(* CODESYS project untitled1.library
   Placeholder: TwinCAT_LIB
   Title: TwinCAT_LIB
   Version: 1.65
   Description: Baisc library's for s88 programming
   Company: Farnwood Engineering

Project tree, tasks and I/O mapping:
  libraries: Tc2_Standard, * (Beckhoff Automation GmbH); Tc2_System, * (Beckhoff Automation GmbH); Tc3_Module, * (Beckhoff Automation GmbH)
  DUTs/
  GVLs/
    POUs/
      LIB/
        1. Control Modules/
          1. DEV_Base/
            function block FB_DeviceBase [ST]
            data type stDevBase
          2. DEV_AnaIn/
            function block FB_DEV_AnaIn [ST]
            interface ITF_DEV_AnaIn
          3. DEV_DigIn/
            function block FB_DEV_DigIn [ST]: FB_init, Force, ResetForce, ActualValue, FallingEdge, RisingEdge
            interface ITF_DigIn: FB_init, Force, ResetForce, ActualValue, FallingEdge, RisingEdge
          4. DEV_Valve/
            ENUMs/
              data type E_ValveState
            STRUCTs/
              data type stDevValve
            function block DEV_Valve [ST]: _FExceptions, _StHmi, Close, Open, Reset, SetMode, ActualState, EmergencyStatus, OperatingMode
            interface ITF_Valve: Close, Open, Reset, SetMode, ActualState, EmergencyStatus, OperatingMode
          5. DEV_ControlValve/
            ENUMs/
              data type E_CtrlValveState
            STRUCTs/
            function block DEV_CtrlValve [ST]: EmergencyStatus, OperatingMode, OutputValue, Reset, SetMode, SetValue
            interface ITF_ControlValve: Reset, SetMode, SetValue, EmergencyStatus, OperatingMode, OutputValue
          6. DEV_Motor/
            ENUMs/
              data type E_MotorState
            STRUCTs/
            interface ITF_Motor: Auto, Manueel, Reset, Richting_L, Richting_R, Start, Stop, Toerental, ActualState, Error_State, State
          7. DEV_ControlMotor/
          ENUMs/
            data type E_OperationMode
          function block FB_Devices [ST]
        2. Equipment Modules/
          1. FB_Base/
            function block FB_EMbase [ST]
            data type stEMbase
          2. EM_Machine_PackML/
            data type E_State_PackML
            function block FB_Machine_PackML [ST]: Abort, Aborting_SC, Clear, Clearing_SC, Completing_SC, Execute_SC, Hold, Holding_SC, Reset, Resetting_SC, Start, Starting_SC, Stop, Stopping_SC, Suspend, Suspending_SC, Unhold, Unholding_SC, Unsuspend, Unsuspending_SC, State, FB_init, ZeroAllVar
            interface ITF_PackML: Abort, Aborting_SC, Clear, Clearing_SC, Completing_SC, Execute_SC, Hold, Holding_SC, Reset, Resetting_SC, Start, Starting_SC, Stop, Stopping_SC, Suspend, Suspending_SC, Unhold, Unholding_SC, Unsuspend, Unsuspending_SC, ZeroAllVar, State, FB_init
            data type STRUCT_Machine_PackML
          2. EM_Transport/
            Enums/
            Structs/
              1. CS/
                data type EM_Transport_CS
              2. HMI/
                data type EM_Transport_HMI
              3. STS/
                data type EM_Transport_STS
              4. ALM/
                data type EM_Transport_ALM
              5. WRN/
                data type EM_Transport_WRN
              6. PAR/
                data type EM_Transport_PAR
              7. SIM/
                data type EM_Transport_SIM
              data type STRUCT_EM_Transport
            function block EM_Transport [ST]: Abort, Clear, Reset, Start, Stop, Auto, Manueel, RPM, State, Tag, ZeroAllVar
            interface ITF_EM_Transport: Abort, Reset, Start, Stop, Auto, Manueel, RPM, State, Tag, ZeroAllVar
          3. EM_Transport_Mechanische_Stop/
            Enums/
              data type E_Mechanische_Stop
            Structs/
              1. CS/
                data type EM_Transport_Mechanische_Stop_CS
              2. HMI/
                data type EM_Transport_Mechanische_Stop_HMI
              3. STS/
                data type EM_Transport_Mechanische_Stop_STS
              4. ALM/
                data type EM_Transport_Mechanische_Stop_ALM
              5. WRN/
                data type EM_Transport_Mechanische_Stop_WRN
              6. PAR/
                data type EM_Transport_Mechanische_Stop_PAR
              7. SIM/
                data type EM_Transport_Mechanische_Stop_SIM
              data type STRUCT_EM_Mechanische_Stop
            function block EM_Transport_Mechanische_Stop [ST]: Close, Open, Stop_State, ZeroAllValues
            interface ITF_EM_Transport_Mechanische_Stop: Close, Open, Stop_State, ZeroAllValues
        3. Units/
          1. UN_Base/
            function block FB_UN_base [ST]
            data type stUNbase
        4. Management layer/
          FB_Alarmhandler/
        FUN/
          function PackML [ST]
          data type STRUCT_PackML
      program MAIN [ST]
  Version/
    global variables Global_Version
  VISUs/
*)

// GVLs/POUs/LIB/1. Control Modules/1. DEV_Base/stDevBase
TYPE stDevBase :
STRUCT
	sTagName : STRING;
	sDescription : STRING;
END_STRUCT
END_TYPE

// GVLs/POUs/LIB/1. Control Modules/4. DEV_Valve/ENUMs/E_ValveState
{attribute 'qualified_only'}
{attribute 'strict'}
TYPE E_ValveState :
(
	Unknown := 0,
	Open := 1,
	Closed := 2,
	Opening := 3,
	Closing := 4,
	Error := -1
);
END_TYPE

// GVLs/POUs/LIB/1. Control Modules/4. DEV_Valve/STRUCTs/stDevValve
TYPE stDevValve :
STRUCT
	//Input to HMI
	bGetHmiError : BOOL;  //True = error
	bGetHmiStatus : BOOL; //True = Open || False = Closed
	eGetState : E_ValveState;
	eGetMode : E_OperationMode;
	
	//Output from HMI
	eSetMode : E_OperationMode; 
END_STRUCT
END_TYPE

// GVLs/POUs/LIB/1. Control Modules/5. DEV_ControlValve/ENUMs/E_CtrlValveState
{attribute 'qualified_only'}
{attribute 'strict'}
TYPE E_CtrlValveState :
(
	Unknown := 0,
	InPosition := 1,
	Moving := 2,
	Error := -1
);
END_TYPE

// GVLs/POUs/LIB/1. Control Modules/6. DEV_Motor/ENUMs/E_MotorState
{attribute 'qualified_only'}
{attribute 'strict'}
TYPE E_MotorState :
(
	Unknown := 0,
	Running := 1,
	Stalled := 2,
	SpeedingUp := 3,
	SpeedingDown := 4,
	Error := -1
);
END_TYPE

// GVLs/POUs/LIB/1. Control Modules/ENUMs/E_OperationMode
{attribute 'qualified_only'}
{attribute 'strict'}
TYPE E_OperationMode :
(
	Off := 0,
	Manual := 1,
	Automatic := 2
);
END_TYPE

// GVLs/POUs/LIB/2. Equipment Modules/1. FB_Base/stEMbase
TYPE stEMbase :
STRUCT
	sTagName : STRING;
	sDescription : STRING;
END_STRUCT
END_TYPE

// GVLs/POUs/LIB/2. Equipment Modules/2. EM_Machine_PackML/E_State_PackML
{attribute 'qualified_only'}
{attribute 'strict'}
TYPE E_State_PackML :
(
	IDLE	:= 0,
	STARTING,
	EXECUTE,
	COMPLETING,
	COMPLETE,
	RESETTING,
	HOLDING,
	HELD,
	UNHOLDING,
	SUSPENDING,
	SUSPENDED,
	UNSUSPENDING,
	ABORTING,
	ABORTED,
	CLEARING,
	STOPPING,
	STOPPED
);
END_TYPE

// GVLs/POUs/LIB/2. Equipment Modules/2. EM_Machine_PackML/STRUCT_Machine_PackML
TYPE STRUCT_Machine_PackML :
STRUCT
	//Properties
	State 			: E_State_PackML;
	//Methods
   	Abort 			: BOOL;
	Aborting_SC 	: BOOL;
	Clear 			: BOOL;
	Clearing_SC 	: BOOL;
	Execute_SC 		: BOOL;
	Completing_SC	: BOOL;
	Hold 			: BOOL;
	Holding_SC 		: BOOL;
	Reset 			: BOOL;
	Resetting_SC 	: BOOL;
	Start 			: BOOL;
	Starting_SC 	: BOOL;
	Stop 			: BOOL;
	Stopping_SC 	: BOOL;
	Suspend 		: BOOL;
	Suspending_SC 	: BOOL;
	Unhold 			: BOOL;
	Unholding_SC 	: BOOL;
	Unsuspend 		: BOOL;
	Unsuspending_SC : BOOL;
END_STRUCT
END_TYPE

// GVLs/POUs/LIB/2. Equipment Modules/2. EM_Transport/Structs/1. CS/EM_Transport_CS
TYPE EM_Transport_CS :
STRUCT
	Start		: BOOL;
	Stop		: BOOL;
	Reset		: BOOL;
	Abort		: BOOL;
	Auto		: BOOL;
	Manueel		: BOOL;
END_STRUCT
END_TYPE

// GVLs/POUs/LIB/2. Equipment Modules/2. EM_Transport/Structs/2. HMI/EM_Transport_HMI
TYPE EM_Transport_HMI :
STRUCT
	Start		: BOOL;
	Stop		: BOOL;
	Reset		: BOOL;
	Abort		: BOOL;
	Auto		: BOOL;
	Manueel		: BOOL;
END_STRUCT
END_TYPE

// GVLs/POUs/LIB/2. Equipment Modules/2. EM_Transport/Structs/3. STS/EM_Transport_STS
TYPE EM_Transport_STS :
STRUCT
	Tag				: STRING;
	State 			: E_State_PackML;
	Manueel			: BOOL;
	Auto			: BOOL;
END_STRUCT
END_TYPE

// GVLs/POUs/LIB/2. Equipment Modules/2. EM_Transport/Structs/4. ALM/EM_Transport_ALM
TYPE EM_Transport_ALM :
STRUCT
END_STRUCT
END_TYPE

// GVLs/POUs/LIB/2. Equipment Modules/2. EM_Transport/Structs/5. WRN/EM_Transport_WRN
TYPE EM_Transport_WRN :
STRUCT
END_STRUCT
END_TYPE

// GVLs/POUs/LIB/2. Equipment Modules/2. EM_Transport/Structs/6. PAR/EM_Transport_PAR
TYPE EM_Transport_PAR :
STRUCT
END_STRUCT
END_TYPE

// GVLs/POUs/LIB/2. Equipment Modules/2. EM_Transport/Structs/7. SIM/EM_Transport_SIM
TYPE EM_Transport_SIM :
STRUCT
END_STRUCT
END_TYPE

// GVLs/POUs/LIB/2. Equipment Modules/2. EM_Transport/Structs/STRUCT_EM_Transport
TYPE STRUCT_EM_Transport :
STRUCT
	CS	: EM_Transport_CS;
	HMI	: EM_Transport_HMI;
	STS	: EM_Transport_STS;
	ALM	: EM_Transport_ALM;
	WRN	: EM_Transport_WRN;
	PAR	: EM_Transport_PAR;
	SIM	: EM_Transport_SIM;	
END_STRUCT
END_TYPE

// GVLs/POUs/LIB/2. Equipment Modules/3. EM_Transport_Mechanische_Stop/Enums/E_Mechanische_Stop
{attribute 'qualified_only'}
{attribute 'strict'}
TYPE E_Mechanische_Stop :
(
	enum_member := 0
);
END_TYPE

// GVLs/POUs/LIB/2. Equipment Modules/3. EM_Transport_Mechanische_Stop/Structs/1. CS/EM_Transport_Mechanische_Stop_CS
TYPE EM_Transport_Mechanische_Stop_CS :
STRUCT
	Start		: BOOL;
	Stop		: BOOL;
	Reset		: BOOL;
	Abort		: BOOL;
	Auto		: BOOL;
	Manueel		: BOOL;
END_STRUCT
END_TYPE

// GVLs/POUs/LIB/2. Equipment Modules/3. EM_Transport_Mechanische_Stop/Structs/2. HMI/EM_Transport_Mechanische_Stop_HMI
TYPE EM_Transport_Mechanische_Stop_HMI :
STRUCT
	Start		: BOOL;
	Stop		: BOOL;
	Reset		: BOOL;
	Abort		: BOOL;
	Auto		: BOOL;
	Manueel		: BOOL;
END_STRUCT
END_TYPE

// GVLs/POUs/LIB/2. Equipment Modules/3. EM_Transport_Mechanische_Stop/Structs/3. STS/EM_Transport_Mechanische_Stop_STS
TYPE EM_Transport_Mechanische_Stop_STS :
STRUCT
	Tag				: STRING;
	State 			: E_Mechanische_Stop;
	Manueel			: BOOL;
	Auto			: BOOL;
END_STRUCT
END_TYPE

// GVLs/POUs/LIB/2. Equipment Modules/3. EM_Transport_Mechanische_Stop/Structs/4. ALM/EM_Transport_Mechanische_Stop_ALM
TYPE EM_Transport_Mechanische_Stop_ALM :
STRUCT
END_STRUCT
END_TYPE

// GVLs/POUs/LIB/2. Equipment Modules/3. EM_Transport_Mechanische_Stop/Structs/5. WRN/EM_Transport_Mechanische_Stop_WRN
TYPE EM_Transport_Mechanische_Stop_WRN :
STRUCT
END_STRUCT
END_TYPE

// GVLs/POUs/LIB/2. Equipment Modules/3. EM_Transport_Mechanische_Stop/Structs/6. PAR/EM_Transport_Mechanische_Stop_PAR
TYPE EM_Transport_Mechanische_Stop_PAR :
STRUCT
END_STRUCT
END_TYPE

// GVLs/POUs/LIB/2. Equipment Modules/3. EM_Transport_Mechanische_Stop/Structs/7. SIM/EM_Transport_Mechanische_Stop_SIM
TYPE EM_Transport_Mechanische_Stop_SIM :
STRUCT
END_STRUCT
END_TYPE

// GVLs/POUs/LIB/2. Equipment Modules/3. EM_Transport_Mechanische_Stop/Structs/STRUCT_EM_Mechanische_Stop
TYPE STRUCT_EM_Mechanische_Stop :
STRUCT
	CS	: EM_Transport_Mechanische_Stop_CS;
	HMI	: EM_Transport_Mechanische_Stop_HMI;
	STS	: EM_Transport_Mechanische_Stop_STS;
	ALM	: EM_Transport_Mechanische_Stop_ALM;
	WRN	: EM_Transport_Mechanische_Stop_WRN;
	PAR	: EM_Transport_Mechanische_Stop_PAR;
	SIM	: EM_Transport_Mechanische_Stop_SIM;	
END_STRUCT
END_TYPE

// GVLs/POUs/LIB/3. Units/1. UN_Base/stUNbase
TYPE stUNbase :
STRUCT
	sTagName : STRING;
	sDescription : STRING;
END_STRUCT
END_TYPE

// GVLs/POUs/LIB/FUN/STRUCT_PackML
TYPE STRUCT_PackML :
STRUCT
	State 			: E_State_PackML;
   	Abort 			: BOOL;
	Aborting_SC 	: BOOL;
	Clear 			: BOOL;
	Clearing_SC 	: BOOL;
	Execute_SC 		: BOOL;
	Completing_SC	: BOOL;
	Hold 			: BOOL;
	Holding_SC 		: BOOL;
	Reset 			: BOOL;
	Resetting_SC 	: BOOL;
	Start 			: BOOL;
	Starting_SC 	: BOOL;
	Stop 			: BOOL;
	Stopping_SC 	: BOOL;
	Suspend 		: BOOL;
	Suspending_SC 	: BOOL;
	Unhold 			: BOOL;
	Unholding_SC 	: BOOL;
	Unsuspend 		: BOOL;
	Unsuspending_SC : BOOL;
END_STRUCT
END_TYPE

// Version/Global_Version
{attribute 'TcGenerated'}
{attribute 'no-analysis'}
{attribute 'linkalways'}
// This function has been automatically generated from the project information.
VAR_GLOBAL CONSTANT
	{attribute 'const_non_replaced'}
	stLibVersion_TwinCAT_LIB : ST_LibVersion := (iMajor := 1, iMinor := 65, iBuild := 0, iRevision := 0, nFlags := 0, sVersion := '1.65');
END_VAR

// GVLs/POUs/LIB/1. Control Modules/1. DEV_Base/FB_DeviceBase
FUNCTION_BLOCK FB_DeviceBase
VAR
	TagName : STRING;
	Description : STRING;
	TagID : INT;
END_VAR

END_FUNCTION_BLOCK

// GVLs/POUs/LIB/1. Control Modules/2. DEV_AnaIn/FB_DEV_AnaIn
FUNCTION_BLOCK FB_DEV_AnaIn EXTENDS FB_DeviceBase IMPLEMENTS ITF_DEV_AnaIn
VAR_INPUT
END_VAR
VAR_OUTPUT
END_VAR
VAR
END_VAR

END_FUNCTION_BLOCK

// GVLs/POUs/LIB/1. Control Modules/2. DEV_AnaIn/ITF_DEV_AnaIn
INTERFACE ITF_DEV_AnaIn

END_INTERFACE

// GVLs/POUs/LIB/1. Control Modules/3. DEV_DigIn/FB_DEV_DigIn
FUNCTION_BLOCK FB_DEV_DigIn EXTENDS FB_DeviceBase IMPLEMENTS ITF_DigIn
VAR
	
END_VAR

{warning 'add method implementation '}
METHOD FB_init : BOOL
VAR_INPUT
	(* if TRUE, the retain variables are initialized (warm start / cold start)*)
	bInitRetains	: BOOL;
	(* if TRUE, the instance afterwards gets moved into the copy code (online change)*)
	bInCopyCode	: BOOL;
END_VAR
END_METHOD

{warning 'add method implementation '}
METHOD Force : BOOL
VAR_INPUT
	ForceValue	: BOOL;
END_VAR
END_METHOD

{warning 'add method implementation '}
METHOD ResetForce : BOOL
END_METHOD

{warning 'add property implementation'}
PROPERTY ActualValue : BOOL
GET
END_GET
SET
END_SET
END_PROPERTY

{warning 'add property implementation'}
PROPERTY FallingEdge : BOOL
GET
END_GET
SET
END_SET
END_PROPERTY

{warning 'add property implementation'}
PROPERTY RisingEdge : BOOL
GET
END_GET
SET
END_SET
END_PROPERTY

END_FUNCTION_BLOCK

// GVLs/POUs/LIB/1. Control Modules/3. DEV_DigIn/ITF_DigIn
INTERFACE ITF_DigIn

METHOD FB_init : BOOL
VAR_INPUT
	bInitRetains : BOOL; // if TRUE, the retain variables are initialized (warm start / cold start)
	bInCopyCode : BOOL;  // if TRUE, the instance afterwards gets moved into the copy code (online change)
END_VAR
END_METHOD

METHOD Force : BOOL
VAR_INPUT
	ForceValue : BOOL;
END_VAR
END_METHOD

METHOD ResetForce : BOOL
VAR_INPUT
END_VAR
END_METHOD

PROPERTY ActualValue : BOOL
GET
END_GET
SET
END_SET
END_PROPERTY

PROPERTY FallingEdge : BOOL
GET
END_GET
SET
END_SET
END_PROPERTY

PROPERTY RisingEdge : BOOL
GET
END_GET
SET
END_SET
END_PROPERTY

END_INTERFACE

// GVLs/POUs/LIB/1. Control Modules/4. DEV_Valve/DEV_Valve
FUNCTION_BLOCK DEV_Valve EXTENDS FB_DeviceBase IMPLEMENTS ITF_Valve

VAR
	I_FeedbackOpen		AT	%I* : BOOL;
	I_FeedbackClosed 	AT 	%I* : BOOL;
	I_Estop				AT	%I*	: BOOL;
	Q_ValveOutput		AT	%Q*	: BOOL;
	
	s_eActualState				: E_ValveState;
	s_eOperatingMode			: E_OperationMode;
	s_tonFeedbackTime			: TON;
	
	bFeedbackError		: BOOL;
	bEstopActive		: BOOL;
	bBothFeedback		: BOOL;
END_VAR

METHOD _FExceptions : BOOL
VAR_INPUT
END_VAR
END_METHOD

METHOD PRIVATE _StHmi
VAR_INPUT
	stHMI : stDevValve;
END_VAR
END_METHOD

{warning 'add method implementation '}
METHOD Close : BOOL
END_METHOD

{warning 'add method implementation '}
METHOD Open : BOOL
END_METHOD

{warning 'add method implementation '}
METHOD Reset : BOOL
END_METHOD

{warning 'add method implementation '}
METHOD SetMode : BOOL
END_METHOD

{warning 'add property implementation'}
PROPERTY ActualState : E_ValveState
GET
END_GET
END_PROPERTY

{warning 'add property implementation'}
PROPERTY EmergencyStatus : BOOL
GET
END_GET
END_PROPERTY

{warning 'add property implementation'}
PROPERTY OperatingMode : BOOL
GET
END_GET
END_PROPERTY

END_FUNCTION_BLOCK

// GVLs/POUs/LIB/1. Control Modules/4. DEV_Valve/ITF_Valve
INTERFACE ITF_Valve

METHOD Close : BOOL
VAR_INPUT
END_VAR
END_METHOD

METHOD Open : BOOL
VAR_INPUT
END_VAR
END_METHOD

METHOD Reset : BOOL
VAR_INPUT
END_VAR
END_METHOD

METHOD SetMode : BOOL
VAR_INPUT
END_VAR
END_METHOD

PROPERTY ActualState : E_ValveState
GET
END_GET
END_PROPERTY

PROPERTY EmergencyStatus : BOOL
GET
END_GET
END_PROPERTY

PROPERTY OperatingMode : BOOL
GET
END_GET
END_PROPERTY

END_INTERFACE

// GVLs/POUs/LIB/1. Control Modules/5. DEV_ControlValve/DEV_CtrlValve
FUNCTION_BLOCK DEV_CtrlValve EXTENDS FB_DeviceBase IMPLEMENTS ITF_ControlValve
VAR_INPUT
END_VAR
VAR_OUTPUT
END_VAR
VAR
END_VAR

{warning 'add property implementation'}
PROPERTY EmergencyStatus : BOOL
GET
END_GET
END_PROPERTY

{warning 'add property implementation'}
PROPERTY OperatingMode : BOOL
GET
END_GET
END_PROPERTY

{warning 'add property implementation'}
PROPERTY OutputValue : REAL
GET
END_GET
END_PROPERTY

{warning 'add method implementation '}
METHOD Reset : BOOL
END_METHOD

{warning 'add method implementation '}
METHOD SetMode : BOOL
END_METHOD

{warning 'add method implementation '}
METHOD SetValue : BOOL
END_METHOD

END_FUNCTION_BLOCK

// GVLs/POUs/LIB/1. Control Modules/5. DEV_ControlValve/ITF_ControlValve
INTERFACE ITF_ControlValve

METHOD Reset : BOOL
VAR_INPUT
END_VAR
END_METHOD

METHOD SetMode : BOOL
VAR_INPUT
END_VAR
END_METHOD

METHOD SetValue : BOOL
VAR_INPUT
END_VAR
END_METHOD

PROPERTY EmergencyStatus : BOOL
GET
END_GET
END_PROPERTY

PROPERTY OperatingMode : BOOL
GET
END_GET
END_PROPERTY

PROPERTY OutputValue : REAL
GET
END_GET
END_PROPERTY

END_INTERFACE

// GVLs/POUs/LIB/1. Control Modules/6. DEV_Motor/ITF_Motor
INTERFACE ITF_Motor

METHOD Auto : BOOL
VAR_INPUT
END_VAR
END_METHOD

METHOD Manueel : BOOL
VAR_INPUT
END_VAR
END_METHOD

METHOD Reset : BOOL
VAR_INPUT
END_VAR
END_METHOD

METHOD Richting_L : BOOL
VAR_INPUT
END_VAR
END_METHOD

METHOD Richting_R : BOOL
VAR_INPUT
END_VAR
END_METHOD

METHOD Start : BOOL
VAR_INPUT
END_VAR
END_METHOD

METHOD Stop : BOOL
VAR_INPUT
END_VAR
END_METHOD

METHOD Toerental : INT
VAR_INPUT
END_VAR
END_METHOD

PROPERTY ActualState : BOOL
GET
END_GET
END_PROPERTY

PROPERTY Error_State : BOOL
GET
END_GET
END_PROPERTY

PROPERTY State : E_MotorState
GET
END_GET
END_PROPERTY

END_INTERFACE

// GVLs/POUs/LIB/1. Control Modules/FB_Devices
FUNCTION_BLOCK FB_Devices
VAR
	devValveV2012 : DEV_Valve := (TagName := 'V2012', Description := 'Standard Valve', TagID := 1);
	devValveV2020 : DEV_Valve := (TagName := 'V2020', Description := 'Standard Valve', TagID := 2);
	devValveV2021 : DEV_Valve := (TagName := 'V2021', Description := 'Standard Valve', TagID := 3);
	devValveV2022 : DEV_Valve := (TagName := 'V2022', Description := 'Standard Valve', TagID := 4);
END_VAR

devValveV2012();
devValveV2020();
devValveV2021();
devValveV2020();

END_FUNCTION_BLOCK

// GVLs/POUs/LIB/2. Equipment Modules/1. FB_Base/FB_EMbase
FUNCTION_BLOCK FB_EMbase
VAR
	TagName : STRING;
	Description : STRING;
	TagID : INT;
END_VAR

END_FUNCTION_BLOCK

// GVLs/POUs/LIB/2. Equipment Modules/2. EM_Machine_PackML/FB_Machine_PackML
FUNCTION_BLOCK FB_Machine_PackML IMPLEMENTS ITF_PackML
VAR
	fbPackML_mem : STRUCT_Machine_PackML;
END_VAR

(*
$$$$$$$$\                                                                   $$\       $$$$$$$$\                     $$\                                         $$\                     
$$  _____|                                                                  $$ |      $$  _____|                    \__|                                        \__|                    
$$ |   $$$$$$\   $$$$$$\  $$$$$$$\  $$\  $$\  $$\  $$$$$$\   $$$$$$\   $$$$$$$ |      $$ |      $$$$$$$\   $$$$$$\  $$\ $$$$$$$\   $$$$$$\   $$$$$$\   $$$$$$\  $$\ $$$$$$$\   $$$$$$\  
$$$$$\ \____$$\ $$  __$$\ $$  __$$\ $$ | $$ | $$ |$$  __$$\ $$  __$$\ $$  __$$ |      $$$$$\    $$  __$$\ $$  __$$\ $$ |$$  __$$\ $$  __$$\ $$  __$$\ $$  __$$\ $$ |$$  __$$\ $$  __$$\ 
$$  __|$$$$$$$ |$$ |  \__|$$ |  $$ |$$ | $$ | $$ |$$ /  $$ |$$ /  $$ |$$ /  $$ |      $$  __|   $$ |  $$ |$$ /  $$ |$$ |$$ |  $$ |$$$$$$$$ |$$$$$$$$ |$$ |  \__|$$ |$$ |  $$ |$$ /  $$ |
$$ |  $$  __$$ |$$ |      $$ |  $$ |$$ | $$ | $$ |$$ |  $$ |$$ |  $$ |$$ |  $$ |      $$ |      $$ |  $$ |$$ |  $$ |$$ |$$ |  $$ |$$   ____|$$   ____|$$ |      $$ |$$ |  $$ |$$ |  $$ |
$$ |  \$$$$$$$ |$$ |      $$ |  $$ |\$$$$$\$$$$  |\$$$$$$  |\$$$$$$  |\$$$$$$$ |      $$$$$$$$\ $$ |  $$ |\$$$$$$$ |$$ |$$ |  $$ |\$$$$$$$\ \$$$$$$$\ $$ |      $$ |$$ |  $$ |\$$$$$$$ |
\__|   \_______|\__|      \__|  \__| \_____\____/  \______/  \______/  \_______|      \________|\__|  \__| \____$$ |\__|\__|  \__| \_______| \_______|\__|      \__|\__|  \__| \____$$ |
                                                                                                          $$\   $$ |                                                          $$\   $$ |
                                                                                                          \$$$$$$  |                                                          \$$$$$$  |
                                                                                                           \______/                                                            \______/ 
*)

CASE fbPackML_mem.State OF
	E_State_PackML.IDLE 			: 
		//HAPPY FLOW		
		IF fbPackML_mem.Start AND NOT fbPackML_mem.Abort THEN
			fbPackML_mem.State:= E_State_PackML.STARTING;
		END_IF
		
		//EXEPTION HANDLING
		IF fbPackML_mem.Abort THEN
			fbPackML_mem.State:= E_State_PackML.ABORTING;
		END_IF
		IF fbPackML_mem.Stop THEN
			fbPackML_mem.State:= E_State_PackML.STOPPING;
		END_IF
	
	E_State_PackML.STARTING 		:
		//HAPPY FLOW		
		IF fbPackML_mem.Starting_SC AND NOT fbPackML_mem.Abort THEN
			fbPackML_mem.State:= E_State_PackML.IDLE;
		END_IF
		
		//EXEPTION HANDLING
		IF fbPackML_mem.Abort THEN
			fbPackML_mem.State:= E_State_PackML.ABORTING;
		END_IF
		IF fbPackML_mem.Stop THEN
			fbPackML_mem.State:= E_State_PackML.STOPPING;
		END_IF
	
	E_State_PackML.EXECUTE 			: 
		//HAPPY FLOW		
		IF fbPackML_mem.Execute_SC AND NOT fbPackML_mem.Abort THEN
			fbPackML_mem.State:= E_State_PackML.IDLE;
		END_IF
		
		IF fbPackML_mem.Hold THEN
			fbPackML_mem.State:= E_State_PackML.HOLDING;
		END_IF
		
		IF fbPackML_mem.Suspend THEN
			fbPackML_mem.State:= E_State_PackML.SUSPENDED;
		END_IF
		
		//EXEPTION HANDLING
		IF fbPackML_mem.Abort THEN
			fbPackML_mem.State:= E_State_PackML.ABORTING;
		END_IF
		IF fbPackML_mem.Stop THEN
			fbPackML_mem.State:= E_State_PackML.STOPPING;
		END_IF
	
	E_State_PackML.COMPLETE 		:
		//HAPPY FLOW
		fbPackML_mem.State:= E_State_PackML.RESETTING;
	
	E_State_PackML.RESETTING 		:
		//HAPPY FLOW		
		IF fbPackML_mem.Resetting_SC AND NOT fbPackML_mem.Abort THEN
			fbPackML_mem.State:= E_State_PackML.IDLE;
		END_IF
		
		//EXEPTION HANDLING
		IF fbPackML_mem.Abort THEN
			fbPackML_mem.State:= E_State_PackML.ABORTING;
		END_IF
		IF fbPackML_mem.Stop THEN
			fbPackML_mem.State:= E_State_PackML.STOPPING;
		END_IF
	
	E_State_PackML.HOLDING 			:
		//HAPPY FLOW		
		IF fbPackML_mem.Holding_SC AND NOT fbPackML_mem.Abort THEN
			fbPackML_mem.State:= E_State_PackML.HELD;
		END_IF
		
		//EXEPTION HANDLING
		IF fbPackML_mem.Abort THEN
			fbPackML_mem.State:= E_State_PackML.ABORTING;
		END_IF
		IF fbPackML_mem.Stop THEN
			fbPackML_mem.State:= E_State_PackML.STOPPING;
		END_IF
		
	
	E_State_PackML.HELD 			:
		//HAPPY FLOW		
		IF fbPackML_mem.Unhold AND NOT fbPackML_mem.Abort THEN
			fbPackML_mem.State:= E_State_PackML.UNHOLDING;
		END_IF
		
		//EXEPTION HANDLING
		IF fbPackML_mem.Abort THEN
			fbPackML_mem.State:= E_State_PackML.ABORTING;
		END_IF
		IF fbPackML_mem.Stop THEN
			fbPackML_mem.State:= E_State_PackML.STOPPING;
		END_IF
	
	E_State_PackML.UNHOLDING 		:
		//HAPPY FLOW		
		IF fbPackML_mem.Unholding_SC AND NOT fbPackML_mem.Abort THEN
			fbPackML_mem.State:= E_State_PackML.EXECUTE;
		END_IF
		
		//EXEPTION HANDLING
		IF fbPackML_mem.Abort THEN
			fbPackML_mem.State:= E_State_PackML.ABORTING;
		END_IF
		IF fbPackML_mem.Stop THEN
			fbPackML_mem.State:= E_State_PackML.STOPPING;
		END_IF
	
	E_State_PackML.SUSPENDING 		:
		//HAPPY FLOW		
		IF fbPackML_mem.Suspending_SC AND NOT fbPackML_mem.Abort THEN
			fbPackML_mem.State:= E_State_PackML.SUSPENDED;
		END_IF
		
		//EXEPTION HANDLING
		IF fbPackML_mem.Abort THEN
			fbPackML_mem.State:= E_State_PackML.ABORTING;
		END_IF
		IF fbPackML_mem.Stop THEN
			fbPackML_mem.State:= E_State_PackML.STOPPING;
		END_IF
	
	
	E_State_PackML.SUSPENDED 		:
		//HAPPY FLOW		
		IF fbPackML_mem.Unsuspend AND NOT fbPackML_mem.Abort THEN
			fbPackML_mem.State:= E_State_PackML.UNSUSPENDING;
		END_IF
		
		//EXEPTION HANDLING
		IF fbPackML_mem.Abort THEN
			fbPackML_mem.State:= E_State_PackML.ABORTING;
		END_IF
		IF fbPackML_mem.Stop THEN
			fbPackML_mem.State:= E_State_PackML.STOPPING;
		END_IF
	
	E_State_PackML.UNSUSPENDING 	:
		//HAPPY FLOW		
		IF fbPackML_mem.Unsuspending_SC AND NOT fbPackML_mem.Abort THEN
			fbPackML_mem.State:= E_State_PackML.EXECUTE;
		END_IF
		
		//EXEPTION HANDLING
		IF fbPackML_mem.Abort THEN
			fbPackML_mem.State:= E_State_PackML.ABORTING;
		END_IF
		IF fbPackML_mem.Stop THEN
			fbPackML_mem.State:= E_State_PackML.STOPPING;
		END_IF
	
	E_State_PackML.ABORTED			:
		//HAPPY FLOW		
		IF fbPackML_mem.Clear THEN
			fbPackML_mem.State:= E_State_PackML.CLEARING;
		END_IF
	
		
	E_State_PackML.ABORTING			:
		//HAPPY FLOW		
		IF fbPackML_mem.Aborting_SC THEN
			fbPackML_mem.State:= E_State_PackML.ABORTED;
		END_IF
	
		
	E_State_PackML.CLEARING 		:
		//HAPPY FLOW		
		IF fbPackML_mem.Clearing_SC THEN
			fbPackML_mem.State:= E_State_PackML.STOPPED;
		END_IF
		
		//EXEPTION HANDLING
		IF fbPackML_mem.Abort THEN
			fbPackML_mem.State:= E_State_PackML.ABORTING;
		END_IF
		
		
	E_State_PackML.STOPPING 		:
		//HAPPY FLOW
		IF fbPackML_mem.Stopping_SC THEN
			fbPackML_mem.State:= E_State_PackML.STOPPED;
		END_IF
		
		//EXEPTION HANDLING
		IF fbPackML_mem.Abort THEN
			fbPackML_mem.State:= E_State_PackML.ABORTING;
		END_IF
		
	
	E_State_PackML.STOPPED 			: 
		//HAPPY FLOW
		IF fbPackML_mem.Reset AND NOT fbPackML_mem.Abort THEN
			fbPackML_mem.State:= E_State_PackML.RESETTING;
		END_IF
		
		//EXEPTION HANDLING
		IF fbPackML_mem.Abort THEN
			fbPackML_mem.State:= E_State_PackML.ABORTING;
		END_IF
		IF fbPackML_mem.Stop THEN
			fbPackML_mem.State:= E_State_PackML.STOPPING;
		END_IF
END_CASE

// Set variables FALSE
fbPackML_mem.Abort 			:= FALSE;
fbPackML_mem.Aborting_SC 	:= FALSE;
fbPackML_mem.Clear 			:= FALSE;
fbPackML_mem.Clearing_SC 	:= FALSE;
fbPackML_mem.Execute_SC 	:= FALSE;
fbPackML_mem.Completing_SC	:= FALSE;
fbPackML_mem.Hold 			:= FALSE;
fbPackML_mem.Holding_SC 	:= FALSE;
fbPackML_mem.Reset 			:= FALSE;
fbPackML_mem.Resetting_SC 	:= FALSE;
fbPackML_mem.Start 			:= FALSE;
fbPackML_mem.Starting_SC 	:= FALSE;
fbPackML_mem.Stop 			:= FALSE;
fbPackML_mem.Stopping_SC 	:= FALSE;
fbPackML_mem.Suspend 		:= FALSE;
fbPackML_mem.Suspending_SC 	:= FALSE;
fbPackML_mem.Unhold 		:= FALSE;
fbPackML_mem.Unholding_SC 	:= FALSE;
fbPackML_mem.Unsuspend 		:= FALSE;

{warning 'add method implementation '}
METHOD Abort : BOOL
fbPackML_mem.Abort := TRUE;
END_METHOD

{warning 'add method implementation '}
METHOD Aborting_SC : BOOL
fbPackML_mem.Aborting_SC := TRUE;
END_METHOD

{warning 'add method implementation '}
METHOD Clear : BOOL
fbPackML_mem.Clear := TRUE;
END_METHOD

{warning 'add method implementation '}
METHOD Clearing_SC : BOOL
fbPackML_mem.Clearing_SC := TRUE;
END_METHOD

{warning 'add method implementation '}
METHOD Completing_SC : BOOL
fbPackML_mem.Completing_SC := TRUE;
END_METHOD

{warning 'add method implementation '}
METHOD Execute_SC : BOOL
fbPackML_mem.Execute_SC := TRUE;
END_METHOD

{warning 'add method implementation '}
METHOD Hold : BOOL
fbPackML_mem.Hold := TRUE;
END_METHOD

{warning 'add method implementation '}
METHOD Holding_SC : BOOL
fbPackML_mem.Holding_SC := TRUE;
END_METHOD

{warning 'add method implementation '}
METHOD Reset : BOOL
fbPackML_mem.Reset := TRUE;
END_METHOD

{warning 'add method implementation '}
METHOD Resetting_SC : BOOL
fbPackML_mem.Resetting_SC := TRUE;
END_METHOD

{warning 'add method implementation '}
METHOD Start : BOOL
fbPackML_mem.Start := TRUE;
END_METHOD

{warning 'add method implementation '}
METHOD Starting_SC : BOOL
fbPackML_mem.Starting_SC := TRUE;
END_METHOD

{warning 'add method implementation '}
METHOD Stop : BOOL
fbPackML_mem.Stop := TRUE;
END_METHOD

{warning 'add method implementation '}
METHOD Stopping_SC : BOOL
fbPackML_mem.Stopping_SC := TRUE;
END_METHOD

{warning 'add method implementation '}
METHOD Suspend : BOOL
fbPackML_mem.Suspend := TRUE;
END_METHOD

{warning 'add method implementation '}
METHOD Suspending_SC : BOOL
fbPackML_mem.Suspending_SC := TRUE;
END_METHOD

{warning 'add method implementation '}
METHOD Unhold : BOOL
fbPackML_mem.Unhold := TRUE;
END_METHOD

{warning 'add method implementation '}
METHOD Unholding_SC : BOOL
fbPackML_mem.Unholding_SC := TRUE;
END_METHOD

{warning 'add method implementation '}
METHOD Unsuspend : BOOL
fbPackML_mem.Unsuspend := TRUE;
END_METHOD

METHOD Unsuspending_SC : BOOL
VAR_INPUT
END_VAR
fbPackML_mem.Unsuspending_SC := TRUE;
END_METHOD

{warning 'add property implementation'}
PROPERTY State : E_State_PackML
GET
State := fbPackML_mem.State;
END_GET
END_PROPERTY

METHOD FB_init : BOOL
VAR_INPUT
    bInitRetains : BOOL; // if TRUE, the retain variables are initialized (warm start / cold start)
    bInCopyCode  : BOOL; // if TRUE, the instance afterwards gets moved into the copy code (online change)
END_VAR
END_METHOD

{warning 'add method implementation '}
METHOD ZeroAllVar : BOOL
fbPackML_mem.Abort				:= FALSE;
fbPackML_mem.Aborting_SC		:= FALSE;
fbPackML_mem.Clear				:= FALSE;
fbPackML_mem.Clearing_SC		:= FALSE;
fbPackML_mem.Completing_SC		:= FALSE;
fbPackML_mem.Execute_SC			:= FALSE;
fbPackML_mem.Hold				:= FALSE;
fbPackML_mem.Holding_SC			:= FALSE;
fbPackML_mem.Reset				:= FALSE;
fbPackML_mem.Resetting_SC		:= FALSE;
fbPackML_mem.Start				:= FALSE;
fbPackML_mem.Starting_SC		:= FALSE;
fbPackML_mem.Stop				:= FALSE;
fbPackML_mem.Stopping_SC		:= FALSE;
fbPackML_mem.Suspend			:= FALSE;
fbPackML_mem.Suspending_SC		:= FALSE;
fbPackML_mem.Unhold				:= FALSE;
fbPackML_mem.Unholding_SC		:= FALSE;
fbPackML_mem.Unsuspend			:= FALSE;
fbPackML_mem.Unsuspending_SC	:= FALSE;
END_METHOD

END_FUNCTION_BLOCK

// GVLs/POUs/LIB/2. Equipment Modules/2. EM_Machine_PackML/ITF_PackML
INTERFACE ITF_PackML

METHOD Abort : BOOL
VAR_INPUT
END_VAR
END_METHOD

METHOD Aborting_SC : BOOL
VAR_INPUT
END_VAR
END_METHOD

METHOD Clear : BOOL
VAR_INPUT
END_VAR
END_METHOD

METHOD Clearing_SC : BOOL
VAR_INPUT
END_VAR
END_METHOD

METHOD Completing_SC : BOOL
VAR_INPUT
END_VAR
END_METHOD

METHOD Execute_SC : BOOL
VAR_INPUT
END_VAR
END_METHOD

METHOD Hold : BOOL
VAR_INPUT
END_VAR
END_METHOD

METHOD Holding_SC : BOOL
VAR_INPUT
END_VAR
END_METHOD

METHOD Reset : BOOL
VAR_INPUT
END_VAR
END_METHOD

METHOD Resetting_SC : BOOL
VAR_INPUT
END_VAR
END_METHOD

METHOD Start : BOOL
VAR_INPUT
END_VAR
END_METHOD

METHOD Starting_SC : BOOL
VAR_INPUT
END_VAR
END_METHOD

METHOD Stop : BOOL
VAR_INPUT
END_VAR
END_METHOD

METHOD Stopping_SC : BOOL
VAR_INPUT
END_VAR
END_METHOD

METHOD Suspend : BOOL
VAR_INPUT
END_VAR
END_METHOD

METHOD Suspending_SC : BOOL
VAR_INPUT
END_VAR
END_METHOD

METHOD Unhold : BOOL
VAR_INPUT
END_VAR
END_METHOD

METHOD Unholding_SC : BOOL
VAR_INPUT
END_VAR
END_METHOD

METHOD Unsuspend : BOOL
VAR_INPUT
END_VAR
END_METHOD

METHOD Unsuspending_SC : BOOL
VAR_INPUT
END_VAR
END_METHOD

METHOD ZeroAllVar : BOOL
VAR_INPUT
END_VAR
END_METHOD

PROPERTY State : E_State_PackML
GET
END_GET
END_PROPERTY

METHOD FB_init : BOOL
VAR_INPUT
	bInitRetains : BOOL; // if TRUE, the retain variables are initialized (warm start / cold start)
	bInCopyCode : BOOL;  // if TRUE, the instance afterwards gets moved into the copy code (online change)
END_VAR
END_METHOD

END_INTERFACE

// GVLs/POUs/LIB/2. Equipment Modules/2. EM_Transport/EM_Transport
FUNCTION_BLOCK EM_Transport IMPLEMENTS  ITF_EM_Transport

VAR
	fb_mem : STRUCT_EM_Transport;
END_VAR

{warning 'add method implementation '}
METHOD Abort : BOOL
END_METHOD

{warning 'add method implementation '}
METHOD Clear : BOOL
END_METHOD

{warning 'add method implementation '}
METHOD Reset : BOOL
END_METHOD

{warning 'add method implementation '}
METHOD Start : BOOL
END_METHOD

{warning 'add method implementation '}
METHOD Stop : BOOL
END_METHOD

PROPERTY Auto : BOOl
GET
AUTO := fb_mem.STS.Auto;
END_GET
SET
fb_mem.CS.Auto := AUTO;
END_SET
END_PROPERTY

PROPERTY Manueel : BOOl
GET
Manueel := fb_mem.STS.Manueel;
END_GET
SET
fb_mem.CS.Manueel :=  Manueel;
END_SET
END_PROPERTY

{warning 'add property implementation'}
PROPERTY RPM : INT
GET
END_GET
SET
END_SET
END_PROPERTY

{warning 'add property implementation'}
PROPERTY State : E_State_PackML
GET
State := fb_mem.STS.State;
END_GET
END_PROPERTY

{warning 'add property implementation'}
PROPERTY Tag : STRING
GET
Tag := fb_mem.STS.Tag;
END_GET
END_PROPERTY

{warning 'add method implementation '}
METHOD ZeroAllVar : BOOL
END_METHOD

END_FUNCTION_BLOCK

// GVLs/POUs/LIB/2. Equipment Modules/2. EM_Transport/ITF_EM_Transport
INTERFACE ITF_EM_Transport

METHOD Abort : BOOL
VAR_INPUT
END_VAR
END_METHOD

METHOD Reset : BOOL
VAR_INPUT
END_VAR
END_METHOD

METHOD Start : BOOL
VAR_INPUT
END_VAR
END_METHOD

METHOD Stop : BOOL
VAR_INPUT
END_VAR
END_METHOD

PROPERTY Auto : BOOL
GET
END_GET
SET
END_SET
END_PROPERTY

PROPERTY Manueel : BOOL
GET
END_GET
SET
END_SET
END_PROPERTY

PROPERTY RPM : INT
GET
END_GET
SET
END_SET
END_PROPERTY

PROPERTY State : E_State_PackML
GET
END_GET
END_PROPERTY

PROPERTY Tag : STRING
GET
END_GET
END_PROPERTY

METHOD ZeroAllVar : BOOL
VAR_INPUT
END_VAR
END_METHOD

END_INTERFACE

// GVLs/POUs/LIB/2. Equipment Modules/3. EM_Transport_Mechanische_Stop/EM_Transport_Mechanische_Stop
FUNCTION_BLOCK EM_Transport_Mechanische_Stop EXTENDS EM_Transport IMPLEMENTS  ITF_EM_Transport_Mechanische_Stop

VAR
	fbMechanischeStop_mem : STRUCT_EM_Mechanische_Stop;
END_VAR

{warning 'add method implementation '}
METHOD Close : BOOL
END_METHOD

{warning 'add method implementation '}
METHOD Open : BOOL
END_METHOD

PROPERTY Stop_State : E_Mechanische_Stop
GET
Stop_State := fbMechanischeStop_mem.STS.State;
END_GET
END_PROPERTY

{warning 'add method implementation '}
METHOD ZeroAllValues : BOOL
END_METHOD

END_FUNCTION_BLOCK

// GVLs/POUs/LIB/2. Equipment Modules/3. EM_Transport_Mechanische_Stop/ITF_EM_Transport_Mechanische_Stop
INTERFACE ITF_EM_Transport_Mechanische_Stop

METHOD Close : BOOL
VAR_INPUT
END_VAR
END_METHOD

METHOD Open : BOOL
VAR_INPUT
END_VAR
END_METHOD

PROPERTY Stop_State : E_Mechanische_Stop
GET
END_GET
END_PROPERTY

METHOD ZeroAllValues : BOOL
VAR_INPUT
END_VAR
END_METHOD

END_INTERFACE

// GVLs/POUs/LIB/3. Units/1. UN_Base/FB_UN_base
FUNCTION_BLOCK FB_UN_base
VAR
	TagName : STRING;
	Description : STRING;
	TagID : INT;
END_VAR

END_FUNCTION_BLOCK

// GVLs/POUs/LIB/FUN/PackML
FUNCTION PackML : E_State_PackML
VAR_INPUT
	Abort 			: BOOL;
	Aborting_SC 	: BOOL;
	Clear 			: BOOL;
	Clearing_SC 	: BOOL;
	Execute_SC 		: BOOL;
	Completing_SC	: BOOL;
	Hold 			: BOOL;
	Holding_SC 		: BOOL;
	Reset 			: BOOL;
	Resetting_SC 	: BOOL;
	Start 			: BOOL;
	Starting_SC 	: BOOL;
	Stop 			: BOOL;
	Stopping_SC 	: BOOL;
	Suspend 		: BOOL;
	Suspending_SC 	: BOOL;
	Unhold 			: BOOL;
	Unholding_SC 	: BOOL;
	Unsuspend 		: BOOL;
	Unsuspending_SC : BOOL;
END_VAR
VAR
	fb_mem			: STRUCT_PackML;
	bFirstCycleBit	: BOOL := FALSE;
END_VAR

(*
$$$$$$$$\                                                                   $$\       $$$$$$$$\                     $$\                                         $$\                     
$$  _____|                                                                  $$ |      $$  _____|                    \__|                                        \__|                    
$$ |   $$$$$$\   $$$$$$\  $$$$$$$\  $$\  $$\  $$\  $$$$$$\   $$$$$$\   $$$$$$$ |      $$ |      $$$$$$$\   $$$$$$\  $$\ $$$$$$$\   $$$$$$\   $$$$$$\   $$$$$$\  $$\ $$$$$$$\   $$$$$$\  
$$$$$\ \____$$\ $$  __$$\ $$  __$$\ $$ | $$ | $$ |$$  __$$\ $$  __$$\ $$  __$$ |      $$$$$\    $$  __$$\ $$  __$$\ $$ |$$  __$$\ $$  __$$\ $$  __$$\ $$  __$$\ $$ |$$  __$$\ $$  __$$\ 
$$  __|$$$$$$$ |$$ |  \__|$$ |  $$ |$$ | $$ | $$ |$$ /  $$ |$$ /  $$ |$$ /  $$ |      $$  __|   $$ |  $$ |$$ /  $$ |$$ |$$ |  $$ |$$$$$$$$ |$$$$$$$$ |$$ |  \__|$$ |$$ |  $$ |$$ /  $$ |
$$ |  $$  __$$ |$$ |      $$ |  $$ |$$ | $$ | $$ |$$ |  $$ |$$ |  $$ |$$ |  $$ |      $$ |      $$ |  $$ |$$ |  $$ |$$ |$$ |  $$ |$$   ____|$$   ____|$$ |      $$ |$$ |  $$ |$$ |  $$ |
$$ |  \$$$$$$$ |$$ |      $$ |  $$ |\$$$$$\$$$$  |\$$$$$$  |\$$$$$$  |\$$$$$$$ |      $$$$$$$$\ $$ |  $$ |\$$$$$$$ |$$ |$$ |  $$ |\$$$$$$$\ \$$$$$$$\ $$ |      $$ |$$ |  $$ |\$$$$$$$ |
\__|   \_______|\__|      \__|  \__| \_____\____/  \______/  \______/  \_______|      \________|\__|  \__| \____$$ |\__|\__|  \__| \_______| \_______|\__|      \__|\__|  \__| \____$$ |
                                                                                                          $$\   $$ |                                                          $$\   $$ |
                                                                                                          \$$$$$$  |                                                          \$$$$$$  |
                                                                                                           \______/                                                            \______/ 
*)
//INPUT NAAR STRUCT
fb_mem.Abort 			:= Abort;
fb_mem.Aborting_SC 		:= Aborting_SC;
fb_mem.Clear 			:= Clear;
fb_mem.Clearing_SC 		:= Clearing_SC;
fb_mem.Execute_SC 		:= Execute_SC;
fb_mem.Completing_SC	:= Completing_SC;
fb_mem.Hold 			:= Hold;
fb_mem.Holding_SC 		:= Holding_SC;
fb_mem.Reset 			:= Reset;
fb_mem.Resetting_SC 	:= Resetting_SC;
fb_mem.Start 			:= Start;
fb_mem.Starting_SC 		:= Starting_SC;
fb_mem.Stop 			:= Stop;
fb_mem.Stopping_SC 		:= Stopping_SC;
fb_mem.Suspend 			:= Suspend;
fb_mem.Suspending_SC 	:= Suspending_SC;
fb_mem.Unhold 			:= Unhold;
fb_mem.Unholding_SC 	:= Unholding_SC;
fb_mem.Unsuspend 		:= Unsuspend;
fb_mem.Unsuspending_SC	:= Unsuspending_SC;

// FIRST CYCLE
IF bFIrstCycleBit THEN
	fb_mem.State := E_State_PackML.RESETTING;
	bFirstCycleBit := TRUE;
END_IF

//TRANSITIES
CASE fb_mem.State OF
	E_State_PackML.IDLE 			: 
		//HAPPY FLOW		
		IF fb_mem.Start AND NOT fb_mem.Abort THEN
			fb_mem.State:= E_State_PackML.STARTING;
		END_IF
		
		//EXEPTION HANDLING
		IF fb_mem.Abort THEN
			fb_mem.State:= E_State_PackML.ABORTING;
		END_IF
		IF fb_mem.Stop THEN
			fb_mem.State:= E_State_PackML.STOPPING;
		END_IF
	
	E_State_PackML.STARTING 		:
		//HAPPY FLOW		
		IF fb_mem.Starting_SC AND NOT fb_mem.Abort THEN
			fb_mem.State:= E_State_PackML.EXECUTE;
		END_IF
		
		//EXEPTION HANDLING
		IF fb_mem.Abort THEN
			fb_mem.State:= E_State_PackML.ABORTING;
		END_IF
		IF fb_mem.Stop THEN
			fb_mem.State:= E_State_PackML.STOPPING;
		END_IF
	
	E_State_PackML.EXECUTE 			: 
		//HAPPY FLOW		
		IF fb_mem.Execute_SC AND NOT fb_mem.Abort THEN
			fb_mem.State:= E_State_PackML.IDLE;
		END_IF
		
		IF fb_mem.Hold THEN
			fb_mem.State:= E_State_PackML.HOLDING;
		END_IF
		
		IF fb_mem.Suspend THEN
			fb_mem.State:= E_State_PackML.SUSPENDED;
		END_IF
		
		//EXEPTION HANDLING
		IF fb_mem.Abort THEN
			fb_mem.State:= E_State_PackML.ABORTING;
		END_IF
		IF fb_mem.Stop THEN
			fb_mem.State:= E_State_PackML.STOPPING;
		END_IF
	
	E_State_PackML.COMPLETE 		:
		//HAPPY FLOW
		fb_mem.State:= E_State_PackML.RESETTING;
	
	E_State_PackML.RESETTING 		:
		//HAPPY FLOW		
		IF fb_mem.Resetting_SC AND NOT fb_mem.Abort THEN
			fb_mem.State:= E_State_PackML.IDLE;
		END_IF
		
		//EXEPTION HANDLING
		IF fb_mem.Abort THEN
			fb_mem.State:= E_State_PackML.ABORTING;
		END_IF
		IF fb_mem.Stop THEN
			fb_mem.State:= E_State_PackML.STOPPING;
		END_IF
	
	E_State_PackML.HOLDING 			:
		//HAPPY FLOW		
		IF fb_mem.Holding_SC AND NOT fb_mem.Abort THEN
			fb_mem.State:= E_State_PackML.HELD;
		END_IF
		
		//EXEPTION HANDLING
		IF fb_mem.Abort THEN
			fb_mem.State:= E_State_PackML.ABORTING;
		END_IF
		IF fb_mem.Stop THEN
			fb_mem.State:= E_State_PackML.STOPPING;
		END_IF
		
	
	E_State_PackML.HELD 			:
		//HAPPY FLOW		
		IF fb_mem.Unhold AND NOT fb_mem.Abort THEN
			fb_mem.State:= E_State_PackML.UNHOLDING;
		END_IF
		
		//EXEPTION HANDLING
		IF fb_mem.Abort THEN
			fb_mem.State:= E_State_PackML.ABORTING;
		END_IF
		IF fb_mem.Stop THEN
			fb_mem.State:= E_State_PackML.STOPPING;
		END_IF
	
	E_State_PackML.UNHOLDING 		:
		//HAPPY FLOW		
		IF fb_mem.Unholding_SC AND NOT fb_mem.Abort THEN
			fb_mem.State:= E_State_PackML.EXECUTE;
		END_IF
		
		//EXEPTION HANDLING
		IF fb_mem.Abort THEN
			fb_mem.State:= E_State_PackML.ABORTING;
		END_IF
		IF fb_mem.Stop THEN
			fb_mem.State:= E_State_PackML.STOPPING;
		END_IF
	
	E_State_PackML.SUSPENDING 		:
		//HAPPY FLOW		
		IF fb_mem.Suspending_SC AND NOT fb_mem.Abort THEN
			fb_mem.State:= E_State_PackML.SUSPENDED;
		END_IF
		
		//EXEPTION HANDLING
		IF fb_mem.Abort THEN
			fb_mem.State:= E_State_PackML.ABORTING;
		END_IF
		IF fb_mem.Stop THEN
			fb_mem.State:= E_State_PackML.STOPPING;
		END_IF
	
	
	E_State_PackML.SUSPENDED 		:
		//HAPPY FLOW		
		IF fb_mem.Unsuspend AND NOT fb_mem.Abort THEN
			fb_mem.State:= E_State_PackML.UNSUSPENDING;
		END_IF
		
		//EXEPTION HANDLING
		IF fb_mem.Abort THEN
			fb_mem.State:= E_State_PackML.ABORTING;
		END_IF
		IF fb_mem.Stop THEN
			fb_mem.State:= E_State_PackML.STOPPING;
		END_IF
	
	E_State_PackML.UNSUSPENDING 	:
		//HAPPY FLOW		
		IF fb_mem.Unsuspending_SC AND NOT fb_mem.Abort THEN
			fb_mem.State:= E_State_PackML.EXECUTE;
		END_IF
		
		//EXEPTION HANDLING
		IF fb_mem.Abort THEN
			fb_mem.State:= E_State_PackML.ABORTING;
		END_IF
		IF fb_mem.Stop THEN
			fb_mem.State:= E_State_PackML.STOPPING;
		END_IF
	
	E_State_PackML.ABORTED			:
		//HAPPY FLOW		
		IF fb_mem.Clear THEN
			fb_mem.State:= E_State_PackML.CLEARING;
		END_IF
	
		
	E_State_PackML.ABORTING			:
		//HAPPY FLOW		
		IF fb_mem.Aborting_SC THEN
			fb_mem.State:= E_State_PackML.ABORTED;
		END_IF
	
		
	E_State_PackML.CLEARING 		:
		//HAPPY FLOW		
		IF fb_mem.Clearing_SC THEN
			fb_mem.State:= E_State_PackML.STOPPED;
		END_IF
		
		//EXEPTION HANDLING
		IF fb_mem.Abort THEN
			fb_mem.State:= E_State_PackML.ABORTING;
		END_IF
		
		
	E_State_PackML.STOPPING 		:
		//HAPPY FLOW
		IF fb_mem.Stopping_SC THEN
			fb_mem.State:= E_State_PackML.STOPPED;
		END_IF
		
		//EXEPTION HANDLING
		IF fb_mem.Abort THEN
			fb_mem.State:= E_State_PackML.ABORTING;
		END_IF
		
	
	E_State_PackML.STOPPED 			: 
		//HAPPY FLOW
		IF fb_mem.Reset AND NOT fb_mem.Abort THEN
			fb_mem.State:= E_State_PackML.RESETTING;
		END_IF
		
		//EXEPTION HANDLING
		IF fb_mem.Abort THEN
			fb_mem.State:= E_State_PackML.ABORTING;
		END_IF
		IF fb_mem.Stop THEN
			fb_mem.State:= E_State_PackML.STOPPING;
		END_IF
END_CASE
PackML := fb_mem.State;

END_FUNCTION

// GVLs/POUs/MAIN
PROGRAM MAIN
VAR
END_VAR

END_PROGRAM
